	X =  325.043  mm,	Y =   -463.962  mm,	Z =   -309.100  mm,
	W =  90.000 deg,	P =   0.000 deg,	R =   90.000 deg
};
P[4144]{
   GP1:
	UF : 0, UT : 6,		CONFIG : 'N U T, 0, 0, 0',
	X =  326.503  mm,	Y =   -464.145  mm,	Z =   -309.000  mm,
	W =  90.000 deg,	P =   0.000 deg,	R =   90.000 deg
};
P[4145]{
   GP1:
	UF : 0, UT : 6,		CONFIG : 'N U T, 0, 0, 0',
	X =  326.408  mm,	Y =   -463.277  mm,	Z =   -309.100  mm,
	W =  90.000 deg,	P =   0.000 deg,	R =   90.000 deg
};
P[4146]{
   GP1:
	UF : 0, UT : 6,		CONFIG : 'N U T, 0, 0, 0',
	X =  327.820  mm,	Y =   -462.995  mm,	Z =   -314.067  mm,
	W =  90.000 deg,	P =   0.000 deg,	R =   90.000 deg
};
P[4147]{
   GP1:
	UF : 0, UT : 6,		CONFIG : 'N U T, 0, 0, 0',
	X =  329.041  mm,	Y =   -462.354  mm,	Z =   -319.718  mm,
	W =  90.000 deg,	P =   0.000 deg,	R =   90.000 deg
};
P[4148]{
   GP1:
	UF : 0, UT : 6,		CONFIG : 'N U T, 0, 0, 0',
	X =  329.280  mm,	Y =   -461.560  mm,	Z =   -309.100  mm,
	W =  90.000 deg,	P =   0.000 deg,	R =   90.000 deg
};
P[4149]{
   GP1:
	UF : 0, UT : 6,		CONFIG : 'N U T, 0, 0, 0',
	X =  330.107  mm,	Y =   -461.147  mm,	Z =   -309.100  mm,
	W =  90.000 deg,	P =   0.000 deg,	R =   90.000 deg
};
P[4150]{
   GP1:
	UF : 0, UT : 6,		CONFIG : 'N U T, 0, 0, 0',
	X =  330.865  mm,	Y =   -460.954  mm,	Z =   -309.100  mm,
	W =  90.000 deg,	P =   0.000 deg,	R =   90.000 deg
};
P[4151]{
   GP1:
	UF : 0, UT : 6,		CONFIG : 'N U T, 0, 0, 0',
	X =  332.067  mm,	Y =   -460.477  mm,	Z =   -309.050  mm,
	W =  90.000 deg,	P =   0.000 deg,	R =   90.000 deg
};
P[4152]{
   GP1:
	UF : 0, UT : 6,		CONFIG : 'N U T, 0, 0, 0',
	X =  333.038  mm,	Y =   -460.052  mm,	Z =   -320.270  mm,
	W =  90.000 deg,	P =   0.000 deg,	R =   90.000 deg
};
P[4153]{
   GP1:
	UF : 0, UT : 6,		CONFIG : 'N U T, 0, 0, 0',
	X =  333.602  mm,	Y =   -459.170  mm,	Z =   -309.000  mm,
	W =  90.000 deg,	P =   0.000 deg,	R =   90.000 deg
};
P[4154]{
   GP1:
	UF : 0, UT : 6,		CONFIG : 'N U T, 0, 0, 0',
	X =  334.380  mm,	Y =   -458.903  mm,	Z =   -318.263  mm,
	W =  90.000 deg,	P =   0.000 deg,	R =   90.000 deg
};
P[4155]{
   GP1:
	UF : 0, UT : 6,		CONFIG : 'N U T, 0, 0, 0',
	X =  335.103  mm,	Y =   -458.639  mm,	Z =   -309.100  mm,
	W =  90.000 deg,	P =   0.000 deg,	R =   90.000 deg
};
P[4156]{
   GP1:
	UF : 0, UT : 6,		CONFIG : 'N U T, 0, 0, 0',
	X =  335.858  mm,	Y =   -457.956  mm,	Z =   -309.100  mm,
	W =  90.000 deg,	P =   0.000 deg,	R =   90.000 deg
};
P[4157]{
   GP1:
	UF : 0, UT : 6,		CONFIG : 'N U T, 0, 0, 0',
	X =  337.562  mm,	Y =   -457.173  mm,	Z =   -309.100  mm,
	W =  90.000 deg,	P =   0.000 deg,	R =   90.000 deg
};
P[4158]{
   GP1:
	UF : 0, UT : 6,		CONFIG : 'N U T, 0, 0, 0',
	X =  338.604  mm,	Y =   -457.010  mm,	Z =   -313.458  mm,
	W =  90.000 deg,	P =   0.000 deg,	R =   90.000 deg
};
P[4159]{
   GP1:
	UF : 0, UT : 6,		CONFIG : 'N U T, 0, 0, 0',
	X =  339.060  mm,	Y =   -455.926  mm,	Z =   -309.100  mm,
	W =  90.000 deg,	P =   0.000 deg,	R =   90.000 deg
};
P[4160]{
   GP1:
	UF : 0, UT : 6,		CONFIG : 'N U T, 0, 0, 0',
	X =  339.781  mm,	Y =   -456.063  mm,	Z =   -325.483  mm,
	W =  90.000 deg,	P =   0.000 deg,	R =   90.000 deg
};
P[4161]{
   GP1:
	UF : 0, UT : 6,		CONFIG : 'N U T, 0, 0, 0',
	X =  340.866  mm,	Y =   -455.653  mm,	Z =   -309.100  mm,
	W =  90.000 deg,	P =   0.000 deg,	R =   90.000 deg
};
P[4162]{
   GP1:
	UF : 0, UT : 6,		CONFIG : 'N U T, 0, 0, 0',
	X =  341.602  mm,	Y =   -454.931  mm,	Z =   -309.100  mm,
	W =  90.000 deg,	P =   0.000 deg,	R =   90.000 deg
};
P[4163]{
   GP1:
	UF : 0, UT : 6,		CONFIG : 'N U T, 0, 0, 0',
	X =  342.495  mm,	Y =   -454.254  mm,	Z =   -309.100  mm,
	W =  90.000 deg,	P =   0.000 deg,	R =   90.000 deg
};
P[4164]{
   GP1:
	UF : 0, UT : 6,		CONFIG : 'N U T, 0, 0, 0',
	X =  343.799  mm,	Y =   -453.794  mm,	Z =   -316.077  mm,
	W =  90.000 deg,	P =   0.000 deg,	R =   90.000 deg
};
P[4165]{
   GP1:
	UF : 0, UT : 6,		CONFIG : 'N U T, 0, 0, 0',
	X =  344.512  mm,	Y =   -453.611  mm,	Z =   -312.115  mm,
	W =  90.000 deg,	P =   0.000 deg,	R =   90.000 deg
};
P[4166]{
   GP1:
	UF : 0, UT : 6,		CONFIG : 'N U T, 0, 0, 0',
	X =  344.893  mm,	Y =   -452.754  mm,	Z =   -309.100  mm,
	W =  90.000 deg,	P =   0.000 deg,	R =   90.000 deg
};
P[4167]{
   GP1:
	UF : 0, UT : 6,		CONFIG : 'N U T, 0, 0, 0',
	X =  345.876  mm,	Y =   -452.177  mm,	Z =   -309.100  mm,
	W =  90.000 deg,	P =   0.000 deg,	R =   90.000 deg
};
P[4168]{
   GP1:
	UF : 0, UT : 6,		CONFIG : 'N U T, 0, 0, 0',
	X =  346.784  mm,	Y =   -451.868  mm,	Z =   -317.158  mm,
	W =  90.000 deg,	P =   0.000 deg,	R =   90.000 deg
};
P[4169]{
   GP1:
	UF : 0, UT : 6,		CONFIG : 'N U T, 0, 0, 0',
	X =  347.518  mm,	Y =   -451.393  mm,	Z =   -309.100  mm,
	W =  90.000 deg,	P =   0.000 deg,	R =   90.000 deg
};
P[4170]{
   GP1:
	UF : 0, UT : 6,		CONFIG : 'N U T, 0, 0, 0',
	X =  348.500  mm,	Y =   -450.922  mm,	Z =   -309.100  mm,
	W =  90.000 deg,	P =   0.000 deg,	R =   90.000 deg
};
P[4171]{
   GP1:
	UF : 0, UT : 6,		CONFIG : 'N U T, 0, 0, 0',
	X =  349.512  mm,	Y =   -449.910  mm,	Z =   -309.100  mm,
	W =  90.000 deg,	P =   0.000 deg,	R =   90.000 deg
};
P[4172]{
   GP1:
	UF : 0, UT : 6,		CONFIG : 'N U T, 0, 0, 0',
	X =  350.498  mm,	Y =   -450.051  mm,	Z =   -317.864  mm,
	W =  90.000 deg,	P =   0.000 deg,	R =   90.000 deg
};
P[4173]{
   GP1:
	UF : 0, UT : 6,		CONFIG : 'N U T, 0, 0, 0',
	X =  351.016  mm,	Y =   -449.580  mm,	Z =   -309.100  mm,
	W =  90.000 deg,	P =   0.000 deg,	R =   90.000 deg
};
P[4174]{
   GP1:
	UF : 0, UT : 6,		CONFIG : 'N U T, 0, 0, 0',
	X =  351.932  mm,	Y =   -448.401  mm,	Z =   -309.100  mm,
	W =  90.000 deg,	P =   0.000 deg,	R =   90.000 deg
};
P[4175]{
   GP1:
	UF : 0, UT : 6,		CONFIG : 'N U T, 0, 0, 0',
	X =  352.880  mm,	Y =   -448.282  mm,	Z =   -309.100  mm,
	W =  90.000 deg,	P =   0.000 deg,	R =   90.000 deg
};
P[4176]{
   GP1:
	UF : 0, UT : 6,		CONFIG : 'N U T, 0, 0, 0',
	X =  353.986  mm,	Y =   -448.251  mm,	Z =   -325.965  mm,
	W =  90.000 deg,	P =   0.000 deg,	R =   90.000 deg
};
P[4177]{
   GP1:
	UF : 0, UT : 6,		CONFIG : 'N U T, 0, 0, 0',
	X =  354.004  mm,	Y =   -447.260  mm,	Z =   -327.146  mm,
	W =  90.000 deg,	P =   0.000 deg,	R =   90.000 deg
};
P[4178]{
   GP1:
	UF : 0, UT : 6,		CONFIG : 'N U T, 0, 0, 0',
	X =  355.173  mm,	Y =   -446.914  mm,	Z =   -309.100  mm,
	W =  90.000 deg,	P =   0.000 deg,	R =   90.000 deg
};
P[4179]{
   GP1:
	UF : 0, UT : 6,		CONFIG : 'N U T, 0, 0, 0',
	X =  356.518  mm,	Y =   -446.536  mm,	Z =   -319.705  mm,
	W =  90.000 deg,	P =   0.000 deg,	R =   90.000 deg
};
P[4180]{
   GP1:
	UF : 0, UT : 6,		CONFIG : 'N U T, 0, 0, 0',
	X =  357.300  mm,	Y =   -445.935  mm,	Z =   -309.000  mm,
	W =  90.000 deg,	P =   0.000 deg,	R =   90.000 deg
};
P[4181]{
   GP1:
	UF : 0, UT : 6,		CONFIG : 'N U T, 0, 0, 0',
	X =  358.004  mm,	Y =   -445.134  mm,	Z =   -309.100  mm,
	W =  90.000 deg,	P =   0.000 deg,	R =   90.000 deg
};
P[4182]{
   GP1:
	UF : 0, UT : 6,		CONFIG : 'N U T, 0, 0, 0',
	X =  359.292  mm,	Y =   -444.664  mm,	Z =   -309.100  mm,
	W =  90.000 deg,	P =   0.000 deg,	R =   90.000 deg
};
P[4183]{
   GP1:
	UF : 0, UT : 6,		CONFIG : 'N U T, 0, 0, 0',
	X =  360.008  mm,	Y =   -444.201  mm,	Z =   -309.000  mm,
	W =  90.000 deg,	P =   0.000 deg,	R =   90.000 deg
};
P[4184]{
   GP1:
	UF : 0, UT : 6,		CONFIG : 'N U T, 0, 0, 0',
	X =  361.188  mm,	Y =   -444.056  mm,	Z =   -325.304  mm,
	W =  90.000 deg,	P =   0.000 deg,	R =   90.000 deg
};
P[4185]{
   GP1:
	UF : 0, UT : 6,		CONFIG : 'N U T, 0, 0, 0',
	X =  361.251  mm,	Y =   -443.010  mm,	Z =   -309.000  mm,
	W =  90.000 deg,	P =   0.000 deg,	R =   90.000 deg
};
P[4186]{
   GP1:
	UF : 0, UT : 6,		CONFIG : 'N U T, 0, 0, 0',
	X =  362.524  mm,	Y =   -443.299  mm,	Z =   -325.248  mm,
	W =  90.000 deg,	P =   0.000 deg,	R =   90.000 deg
};
P[4187]{
   GP1:
	UF : 0, UT : 6,		CONFIG : 'N U T, 0, 0, 0',
	X =  363.226  mm,	Y =   -442.629  mm,	Z =   -327.645  mm,
	W =  90.000 deg,	P =   0.000 deg,	R =   90.000 deg
};
P[4188]{
   GP1:
	UF : 0, UT : 6,		CONFIG : 'N U T, 0, 0, 0',
	X =  363.688  mm,	Y =   -441.945  mm,	Z =   -309.100  mm,
	W =  90.000 deg,	P =   0.000 deg,	R =   90.000 deg
};
P[4189]{
   GP1:
	UF : 0, UT : 6,		CONFIG : 'N U T, 0, 0, 0',
	X =  370.130  mm,	Y =   -455.370  mm,	Z =   -317.842  mm,
	W =  90.000 deg,	P =   0.000 deg,	R =   90.000 deg
};
P[4190]{
   GP1:
	UF : 0, UT : 6,		CONFIG : 'N U T, 0, 0, 0',
	X =  368.313  mm,	Y =   -456.695  mm,	Z =   -320.178  mm,
	W =  90.000 deg,	P =   0.000 deg,	R =   90.000 deg
};
P[4191]{
   GP1:
	UF : 0, UT : 6,		CONFIG : 'N U T, 0, 0, 0',
	X =  367.264  mm,	Y =   -457.201  mm,	Z =   -313.957  mm,
	W =  90.000 deg,	P =   0.000 deg,	R =   90.000 deg
};
P[4192]{
   GP1:
	UF : 0, UT : 6,		CONFIG : 'N U T, 0, 0, 0',
	X =  366.190  mm,	Y =   -457.852  mm,	Z =   -309.100  mm,
	W =  90.000 deg,	P =   0.000 deg,	R =   90.000 deg
};
P[4193]{
   GP1:
	UF : 0, UT : 6,		CONFIG : 'N U T, 0, 0, 0',
	X =  365.352  mm,	Y =   -458.380  mm,	Z =   -323.127  mm,
	W =  90.000 deg,	P =   0.000 deg,	R =   90.000 deg
};
P[4194]{
   GP1:
	UF : 0, UT : 6,		CONFIG : 'N U T, 0, 0, 0',
	X =  364.251  mm,	Y =   -458.803  mm,	Z =   -313.263  mm,
	W =  90.000 deg,	P =   0.000 deg,	R =   90.000 deg
};
P[4195]{
   GP1:
	UF : 0, UT : 6,		CONFIG : 'N U T, 0, 0, 0',
	X =  362.988  mm,	Y =   -459.744  mm,	Z =   -323.904  mm,
	W =  90.000 deg,	P =   0.000 deg,	R =   90.000 deg
};
P[4196]{
   GP1:
	UF : 0, UT : 6,		CONFIG : 'N U T, 0, 0, 0',
	X =  360.054  mm,	Y =   -461.028  mm,	Z =   -309.944  mm,
	W =  90.000 deg,	P =   0.000 deg,	R =   90.000 deg
};
P[4197]{
   GP1:
	UF : 0, UT : 6,		CONFIG : 'N U T, 0, 0, 0',
	X =  359.210  mm,	Y =   -461.622  mm,	Z =   -309.000  mm,
	W =  90.000 deg,	P =   0.000 deg,	R =   90.000 deg
};
P[4198]{
   GP1:
	UF : 0, UT : 6,		CONFIG : 'N U T, 0, 0, 0',
	X =  357.631  mm,	Y =   -462.836  mm,	Z =   -323.003  mm,
	W =  90.000 deg,	P =   0.000 deg,	R =   90.000 deg
};
P[4199]{
   GP1:
	UF : 0, UT : 6,		CONFIG : 'N U T, 0, 0, 0',
	X =  356.113  mm,	Y =   -463.744  mm,	Z =   -321.634  mm,
	W =  90.000 deg,	P =   0.000 deg,	R =   90.000 deg
};
P[4200]{
   GP1:
	UF : 0, UT : 6,		CONFIG : 'N U T, 0, 0, 0',
	X =  353.522  mm,	Y =   -465.245  mm,	Z =   -309.100  mm,
	W =  90.000 deg,	P =   0.000 deg,	R =   90.000 deg
};
P[4201]{
   GP1:
	UF : 0, UT : 6,		CONFIG : 'N U T, 0, 0, 0',
	X =  352.483  mm,	Y =   -465.710  mm,	Z =   -326.795  mm,
	W =  90.000 deg,	P =   0.000 deg,	R =   90.000 deg
};
P[4202]{
   GP1:
	UF : 0, UT : 6,		CONFIG : 'N U T, 0, 0, 0',
	X =  351.674  mm,	Y =   -466.319  mm,	Z =   -318.134  mm,
	W =  90.000 deg,	P =   0.000 deg,	R =   90.000 deg
};
P[4203]{
   GP1:
	UF : 0, UT : 6,		CONFIG : 'N U T, 0, 0, 0',
	X =  350.928  mm,	Y =   -466.372  mm,	Z =   -321.296  mm,
	W =  90.000 deg,	P =   0.000 deg,	R =   90.000 deg
};
P[4204]{
   GP1:
	UF : 0, UT : 6,		CONFIG : 'N U T, 0, 0, 0',
	X =  348.318  mm,	Y =   -468.184  mm,	Z =   -326.716  mm,
	W =  90.000 deg,	P =   0.000 deg,	R =   90.000 deg
};
P[4205]{
   GP1:
	UF : 0, UT : 6,		CONFIG : 'N U T, 0, 0, 0',
	X =  347.496  mm,	Y =   -468.815  mm,	Z =   -311.962  mm,
	W =  90.000 deg,	P =   0.000 deg,	R =   90.000 deg
};
P[4206]{
   GP1:
	UF : 0, UT : 6,		CONFIG : 'N U T, 0, 0, 0',
	X =  346.336  mm,	Y =   -469.289  mm,	Z =   -312.176  mm,
	W =  90.000 deg,	P =   0.000 deg,	R =   90.000 deg
};
P[4207]{
   GP1:
	UF : 0, UT : 6,		CONFIG : 'N U T, 0, 0, 0',
	X =  345.624  mm,	Y =   -469.470  mm,	Z =   -309.000  mm,
	W =  90.000 deg,	P =   0.000 deg,	R =   90.000 deg
};
P[4208]{
   GP1:
	UF : 0, UT : 6,		CONFIG : 'N U T, 0, 0, 0',
	X =  344.976  mm,	Y =   -469.959  mm,	Z =   -312.414  mm,
	W =  90.000 deg,	P =   0.000 deg,	R =   90.000 deg
};
P[4209]{
   GP1:
	UF : 0, UT : 6,		CONFIG : 'N U T, 0, 0, 0',
	X =  344.160  mm,	Y =   -470.743  mm,	Z =   -313.140  mm,
	W =  90.000 deg,	P =   0.000 deg,	R =   90.000 deg
};
P[4210]{
   GP1:
	UF : 0, UT : 6,		CONFIG : 'N U T, 0, 0, 0',
	X =  343.250  mm,	Y =   -471.076  mm,	Z =   -309.000  mm,
	W =  90.000 deg,	P =   0.000 deg,	R =   90.000 deg
};
P[4211]{
   GP1:
	UF : 0, UT : 6,		CONFIG : 'N U T, 0, 0, 0',
	X =  342.335  mm,	Y =   -471.791  mm,	Z =   -309.100  mm,
	W =  90.000 deg,	P =   0.000 deg,	R =   90.000 deg
};
P[4212]{
   GP1:
	UF : 0, UT : 6,		CONFIG : 'N U T, 0, 0, 0',
	X =  341.451  mm,	Y =   -472.238  mm,	Z =   -309.796  mm,
	W =  90.000 deg,	P =   0.000 deg,	R =   90.000 deg
};
P[4213]{
   GP1:
	UF : 0, UT : 6,		CONFIG : 'N U T, 0, 0, 0',
	X =  340.084  mm,	Y =   -473.084  mm,	Z =   -315.122  mm,
	W =  90.000 deg,	P =   0.000 deg,	R =   90.000 deg
};
P[4214]{
   GP1:
	UF : 0, UT : 6,		CONFIG : 'N U T, 0, 0, 0',
	X =  338.651  mm,	Y =   -473.581  mm,	Z =   -314.828  mm,
	W =  90.000 deg,	P =   0.000 deg,	R =   90.000 deg
};
P[4215]{
   GP1:
	UF : 0, UT : 6,		CONFIG : 'N U T, 0, 0, 0',
	X =  337.830  mm,	Y =   -473.912  mm,	Z =   -322.397  mm,
	W =  90.000 deg,	P =   0.000 deg,	R =   90.000 deg
};
P[4216]{
   GP1:
	UF : 0, UT : 6,		CONFIG : 'N U T, 0, 0, 0',
	X =  336.722  mm,	Y =   -474.600  mm,	Z =   -315.900  mm,
	W =  90.000 deg,	P =   0.000 deg,	R =   90.000 deg
};
P[4217]{
   GP1:
	UF : 0, UT : 6,		CONFIG : 'N U T, 0, 0, 0',
	X =  335.536  mm,	Y =   -475.219  mm,	Z =   -309.100  mm,
	W =  90.000 deg,	P =   0.000 deg,	R =   90.000 deg
};
P[4218]{
   GP1:
	UF : 0, UT : 6,		CONFIG : 'N U T, 0, 0, 0',
	X =  334.878  mm,	Y =   -475.959  mm,	Z =   -326.354  mm,
	W =  90.000 deg,	P =   0.000 deg,	R =   90.000 deg
};
P[4219]{
   GP1:
	UF : 0, UT : 6,		CONFIG : 'N U T, 0, 0, 0',
	X =  333.966  mm,	Y =   -476.591  mm,	Z =   -322.102  mm,
	W =  90.000 deg,	P =   0.000 deg,	R =   90.000 deg
};
P[4220]{
   GP1:
	UF : 0, UT : 6,		CONFIG : 'N U T, 0, 0, 0',
	X =  333.254  mm,	Y =   -477.029  mm,	Z =   -309.000  mm,
	W =  90.000 deg,	P =   0.000 deg,	R =   90.000 deg
};
P[4221]{
   GP1:
	UF : 0, UT : 6,		CONFIG : 'N U T, 0, 0, 0',
	X =  330.547  mm,	Y =   -478.456  mm,	Z =   -326.060  mm,
	W =  90.000 deg,	P =   0.000 deg,	R =   90.000 deg
};
P[4222]{
   GP1:
	UF : 0, UT : 6,		CONFIG : 'N U T, 0, 0, 0',
	X =  329.060  mm,	Y =   -479.157  mm,	Z =   -313.599  mm,
	W =  90.000 deg,	P =   0.000 deg,	R =   90.000 deg
};
P[4223]{
   GP1:
	UF : 0, UT : 6,		CONFIG : 'N U T, 0, 0, 0',
	X =  327.871  mm,	Y =   -479.953  mm,	Z =   -311.541  mm,
	W =  90.000 deg,	P =   0.000 deg,	R =   90.000 deg
};
P[4224]{
   GP1:
	UF : 0, UT : 6,		CONFIG : 'N U T, 0, 0, 0',
	X =  327.272  mm,	Y =   -480.484  mm,	Z =   -327.441  mm,
	W =  90.000 deg,	P =   0.000 deg,	R =   90.000 deg
};
P[4225]{
   GP1:
	UF : 0, UT : 6,		CONFIG : 'N U T, 0, 0, 0',
	X =  325.115  mm,	Y =   -481.320  mm,	Z =   -319.370  mm,
	W =  90.000 deg,	P =   0.000 deg,	R =   90.000 deg
};
P[4226]{
   GP1:
	UF : 0, UT : 6,		CONFIG : 'N U T, 0, 0, 0',
	X =  323.945  mm,	Y =   -482.264  mm,	Z =   -323.310  mm,
	W =  90.000 deg,	P =   0.000 deg,	R =   90.000 deg
};
P[4227]{
   GP1:
	UF : 0, UT : 6,		CONFIG : 'N U T, 0, 0, 0',
	X =  323.033  mm,	Y =   -482.925  mm,	Z =   -311.088  mm,
	W =  90.000 deg,	P =   0.000 deg,	R =   90.000 deg
};
P[4228]{
   GP1:
	UF : 0, UT : 6,		CONFIG : 'N U T, 0, 0, 0',
	X =  322.353  mm,	Y =   -483.235  mm,	Z =   -319.952  mm,
	W =  90.000 deg,	P =   0.000 deg,	R =   90.000 deg
};
P[4229]{
   GP1:
	UF : 0, UT : 6,		CONFIG : 'N U T, 0, 0, 0',
	X =  321.581  mm,	Y =   -483.397  mm,	Z =   -309.100  mm,
	W =  90.000 deg,	P =   0.000 deg,	R =   90.000 deg
};
P[4230]{
   GP1:
	UF : 0, UT : 6,		CONFIG : 'N U T, 0, 0, 0',
	X =  320.384  mm,	Y =   -484.322  mm,	Z =   -323.649  mm,
	W =  90.000 deg,	P =   0.000 deg,	R =   90.000 deg
};
P[4231]{
   GP1:
	UF : 0, UT : 6,		CONFIG : 'N U T, 0, 0, 0',
	X =  318.986  mm,	Y =   -485.056  mm,	Z =   -309.000  mm,
	W =  90.000 deg,	P =   0.000 deg,	R =   90.000 deg
};
P[4232]{
   GP1:
	UF : 0, UT : 6,		CONFIG : 'N U T, 0, 0, 0',
	X =  317.976  mm,	Y =   -485.405  mm,	Z =   -321.223  mm,
	W =  90.000 deg,	P =   0.000 deg,	R =   90.000 deg
};
P[4233]{
   GP1:
	UF : 0, UT : 6,		CONFIG : 'N U T, 0, 0, 0',
	X =  317.017  mm,	Y =   -486.084  mm,	Z =   -313.401  mm,
	W =  90.000 deg,	P =   0.000 deg,	R =   90.000 deg
};
P[4234]{
   GP1:
	UF : 0, UT : 6,		CONFIG : 'N U T, 0, 0, 0',
	X =  316.577  mm,	Y =   -486.658  mm,	Z =   -313.931  mm,
	W =  90.000 deg,	P =   0.000 deg,	R =   90.000 deg
};
P[4235]{
   GP1:
	UF : 0, UT : 6,		CONFIG : 'N U T, 0, 0, 0',
	X =  315.204  mm,	Y =   -487.174  mm,	Z =   -318.974  mm,
	W =  90.000 deg,	P =   0.000 deg,	R =   90.000 deg
};
P[4236]{
   GP1:
	UF : 0, UT : 6,		CONFIG : 'N U T, 0, 0, 0',
	X =  314.075  mm,	Y =   -487.965  mm,	Z =   -323.247  mm,
	W =  90.000 deg,	P =   0.000 deg,	R =   90.000 deg
};
P[4237]{
   GP1:
	UF : 0, UT : 6,		CONFIG : 'N U T, 0, 0, 0',
	X =  312.793  mm,	Y =   -488.331  mm,	Z =   -311.315  mm,
	W =  90.000 deg,	P =   0.000 deg,	R =   90.000 deg
};
P[4238]{
   GP1:
	UF : 0, UT : 6,		CONFIG : 'N U T, 0, 0, 0',
	X =  312.228  mm,	Y =   -489.102  mm,	Z =   -311.971  mm,
	W =  90.000 deg,	P =   0.000 deg,	R =   90.000 deg
};
P[4239]{
   GP1:
	UF : 0, UT : 6,		CONFIG : 'N U T, 0, 0, 0',
	X =  311.208  mm,	Y =   -489.769  mm,	Z =   -309.100  mm,
	W =  90.000 deg,	P =   0.000 deg,	R =   90.000 deg
};
P[4240]{
   GP1:
	UF : 0, UT : 6,		CONFIG : 'N U T, 0, 0, 0',
	X =  310.069  mm,	Y =   -490.406  mm,	Z =   -322.968  mm,
	W =  90.000 deg,	P =   0.000 deg,	R =   90.000 deg
};
P[4241]{
   GP1:
	UF : 0, UT : 6,		CONFIG : 'N U T, 0, 0, 0',
	X =  307.990  mm,	Y =   -491.509  mm,	Z =   -309.000  mm,
	W =  90.000 deg,	P =   0.000 deg,	R =   90.000 deg
};
P[4242]{
   GP1:
	UF : 0, UT : 6,		CONFIG : 'N U T, 0, 0, 0',
	X =  307.080  mm,	Y =   -491.884  mm,	Z =   -317.257  mm,
	W =  90.000 deg,	P =   0.000 deg,	R =   90.000 deg
};
P[4243]{
   GP1:
	UF : 0, UT : 6,		CONFIG : 'N U T, 0, 0, 0',
	X =  306.110  mm,	Y =   -492.257  mm,	Z =   -320.855  mm,
	W =  90.000 deg,	P =   0.000 deg,	R =   90.000 deg
};
P[4244]{
   GP1:
	UF : 0, UT : 6,		CONFIG : 'N U T, 0, 0, 0',
	X =  305.486  mm,	Y =   -492.796  mm,	Z =   -324.798  mm,
	W =  90.000 deg,	P =   0.000 deg,	R =   90.000 deg
};
P[4245]{
   GP1:
	UF : 0, UT : 6,		CONFIG : 'N U T, 0, 0, 0',
	X =  304.863  mm,	Y =   -493.261  mm,	Z =   -324.523  mm,
	W =  90.000 deg,	P =   0.000 deg,	R =   90.000 deg
};
P[4246]{
   GP1:
	UF : 0, UT : 6,		CONFIG : 'N U T, 0, 0, 0',
	X =  303.709  mm,	Y =   -493.844  mm,	Z =   -324.912  mm,
	W =  90.000 deg,	P =   0.000 deg,	R =   90.000 deg
};
P[4247]{
   GP1:
	UF : 0, UT : 6,		CONFIG : 'N U T, 0, 0, 0',
	X =  302.792  mm,	Y =   -494.531  mm,	Z =   -309.100  mm,
	W =  90.000 deg,	P =   0.000 deg,	R =   90.000 deg
};
P[4248]{
   GP1:
	UF : 0, UT : 6,		CONFIG : 'N U T, 0, 0, 0',
	X =  301.496  mm,	Y =   -495.214  mm,	Z =   -324.361  mm,
	W =  90.000 deg,	P =   0.000 deg,	R =   90.000 deg
};
P[4249]{
   GP1:
	UF : 0, UT : 6,		CONFIG : 'N U T, 0, 0, 0',
	X =  300.435  mm,	Y =   -495.750  mm,	Z =   -309.000  mm,
	W =  90.000 deg,	P =   0.000 deg,	R =   90.000 deg
};
P[4250]{
   GP1:
	UF : 0, UT : 6,		CONFIG : 'N U T, 0, 0, 0',
	X =  298.649  mm,	Y =   -496.961  mm,	Z =   -312.465  mm,
	W =  90.000 deg,	P =   0.000 deg,	R =   90.000 deg
};
P[4251]{
   GP1:
	UF : 0, UT : 6,		CONFIG : 'N U T, 0, 0, 0',
	X =  297.643  mm,	Y =   -497.369  mm,	Z =   -327.276  mm,
	W =  90.000 deg,	P =   0.000 deg,	R =   90.000 deg
};
P[4252]{
   GP1:
	UF : 0, UT : 6,		CONFIG : 'N U T, 0, 0, 0',
	X =  296.699  mm,	Y =   -497.888  mm,	Z =   -325.030  mm,
	W =  90.000 deg,	P =   0.000 deg,	R =   90.000 deg
};
P[4253]{
   GP1:
	UF : 0, UT : 6,		CONFIG : 'N U T, 0, 0, 0',
	X =  296.076  mm,	Y =   -498.425  mm,	Z =   -317.421  mm,
	W =  90.000 deg,	P =   0.000 deg,	R =   90.000 deg
};
P[4254]{
   GP1:
	UF : 0, UT : 6,		CONFIG : 'N U T, 0, 0, 0',
	X =  295.262  mm,	Y =   -498.510  mm,	Z =   -327.980  mm,
	W =  90.000 deg,	P =   0.000 deg,	R =   90.000 deg
};
P[4255]{
   GP1:
	UF : 0, UT : 6,		CONFIG : 'N U T, 0, 0, 0',
	X =  294.194  mm,	Y =   -499.584  mm,	Z =   -309.568  mm,
	W =  90.000 deg,	P =   0.000 deg,	R =   90.000 deg
};
P[4256]{
   GP1:
	UF : 0, UT : 6,		CONFIG : 'N U T, 0, 0, 0',
	X =  293.467  mm,	Y =   -499.512  mm,	Z =   -323.031  mm,
	W =  90.000 deg,	P =   0.000 deg,	R =   90.000 deg
};
P[4257]{
   GP1:
	UF : 0, UT : 6,		CONFIG : 'N U T, 0, 0, 0',
	X =  291.843  mm,	Y =   -500.658  mm,	Z =   -316.063  mm,
	W =  90.000 deg,	P =   0.000 deg,	R =   90.000 deg
};
P[4258]{
   GP1:
	UF : 0, UT : 6,		CONFIG : 'N U T, 0, 0, 0',
	X =  291.061  mm,	Y =   -501.097  mm,	Z =   -310.941  mm,
	W =  90.000 deg,	P =   0.000 deg,	R =   90.000 deg
};
P[4259]{
   GP1:
	UF : 0, UT : 6,		CONFIG : 'N U T, 0, 0, 0',
	X =  289.807  mm,	Y =   -502.013  mm,	Z =   -317.383  mm,
	W =  90.000 deg,	P =   0.000 deg,	R =   90.000 deg
};
P[4260]{
   GP1:
	UF : 0, UT : 6,		CONFIG : 'N U T, 0, 0, 0',
	X =  289.052  mm,	Y =   -502.193  mm,	Z =   -313.060  mm,
	W =  90.000 deg,	P =   0.000 deg,	R =   90.000 deg
};
P[4261]{
   GP1:
	UF : 0, UT : 6,		CONFIG : 'N U T, 0, 0, 0',
	X =  288.159  mm,	Y =   -503.035  mm,	Z =   -309.000  mm,
	W =  90.000 deg,	P =   0.000 deg,	R =   90.000 deg
};
P[4262]{
   GP1:
	UF : 0, UT : 6,		CONFIG : 'N U T, 0, 0, 0',
	X =  286.879  mm,	Y =   -503.579  mm,	Z =   -327.370  mm,
	W =  90.000 deg,	P =   0.000 deg,	R =   90.000 deg
};
P[4263]{
   GP1:
	UF : 0, UT : 6,		CONFIG : 'N U T, 0, 0, 0',
	X =  285.972  mm,	Y =   -504.314  mm,	Z =   -309.100  mm,
	W =  90.000 deg,	P =   0.000 deg,	R =   90.000 deg
};
P[4264]{
   GP1:
	UF : 0, UT : 6,		CONFIG : 'N U T, 0, 0, 0',
	X =  284.922  mm,	Y =   -504.799  mm,	Z =   -309.000  mm,
	W =  90.000 deg,	P =   0.000 deg,	R =   90.000 deg
};
P[4265]{
   GP1:
	UF : 0, UT : 6,		CONFIG : 'N U T, 0, 0, 0',
	X =  283.518  mm,	Y =   -505.597  mm,	Z =   -324.774  mm,
	W =  90.000 deg,	P =   0.000 deg,	R =   90.000 deg
};
P[4266]{
   GP1:
	UF : 0, UT : 6,		CONFIG : 'N U T, 0, 0, 0',
	X =  281.621  mm,	Y =   -506.363  mm,	Z =   -322.876  mm,
	W =  90.000 deg,	P =   0.000 deg,	R =   90.000 deg
};
P[4267]{
   GP1:
	UF : 0, UT : 6,		CONFIG : 'N U T, 0, 0, 0',
	X =  280.710  mm,	Y =   -507.128  mm,	Z =   -309.000  mm,
	W =  90.000 deg,	P =   0.000 deg,	R =   90.000 deg
};
P[4268]{
   GP1:
	UF : 0, UT : 6,		CONFIG : 'N U T, 0, 0, 0',
	X =  279.612  mm,	Y =   -507.607  mm,	Z =   -319.853  mm,
	W =  90.000 deg,	P =   0.000 deg,	R =   90.000 deg
};
P[4269]{
   GP1:
	UF : 0, UT : 6,		CONFIG : 'N U T, 0, 0, 0',
	X =  278.497  mm,	Y =   -508.589  mm,	Z =   -309.000  mm,
	W =  90.000 deg,	P =   0.000 deg,	R =   90.000 deg
};
P[4270]{
   GP1:
	UF : 0, UT : 6,		CONFIG : 'N U T, 0, 0, 0',
	X =  277.085  mm,	Y =   -509.319  mm,	Z =   -326.506  mm,
	W =  90.000 deg,	P =   0.000 deg,	R =   90.000 deg
};
P[4271]{
   GP1:
	UF : 0, UT : 6,		CONFIG : 'N U T, 0, 0, 0',
	X =  275.580  mm,	Y =   -509.805  mm,	Z =   -309.992  mm,
	W =  90.000 deg,	P =   0.000 deg,	R =   90.000 deg
};
P[4272]{
   GP1:
	UF : 0, UT : 6,		CONFIG : 'N U T, 0, 0, 0',
	X =  274.490  mm,	Y =   -510.823  mm,	Z =   -309.000  mm,
	W =  90.000 deg,	P =   0.000 deg,	R =   90.000 deg
};
P[4273]{
   GP1:
	UF : 0, UT : 6,		CONFIG : 'N U T, 0, 0, 0',
	X =  273.395  mm,	Y =   -511.462  mm,	Z =   -325.321  mm,
	W =  90.000 deg,	P =   0.000 deg,	R =   90.000 deg
};
P[4274]{
   GP1:
	UF : 0, UT : 6,		CONFIG : 'N U T, 0, 0, 0',
	X =  272.390  mm,	Y =   -511.953  mm,	Z =   -327.295  mm,
	W =  90.000 deg,	P =   0.000 deg,	R =   90.000 deg
};
P[4275]{
   GP1:
	UF : 0, UT : 6,		CONFIG : 'N U T, 0, 0, 0',
	X =  271.591  mm,	Y =   -512.486  mm,	Z =   -309.100  mm,
	W =  90.000 deg,	P =   0.000 deg,	R =   90.000 deg
};
P[4276]{
   GP1:
	UF : 0, UT : 6,		CONFIG : 'N U T, 0, 0, 0',
	X =  269.800  mm,	Y =   -513.366  mm,	Z =   -309.730  mm,
	W =  90.000 deg,	P =   0.000 deg,	R =   90.000 deg
};
P[4277]{
   GP1:
	UF : 0, UT : 6,		CONFIG : 'N U T, 0, 0, 0',
	X =  268.979  mm,	Y =   -514.147  mm,	Z =   -325.756  mm,
	W =  90.000 deg,	P =   0.000 deg,	R =   90.000 deg
};
P[4278]{
   GP1:
	UF : 0, UT : 6,		CONFIG : 'N U T, 0, 0, 0',
	X =  267.638  mm,	Y =   -514.775  mm,	Z =   -309.100  mm,
	W =  90.000 deg,	P =   0.000 deg,	R =   90.000 deg
};
P[4279]{
   GP1:
	UF : 0, UT : 6,		CONFIG : 'N U T, 0, 0, 0',
	X =  264.406  mm,	Y =   -516.430  mm,	Z =   -317.911  mm,
	W =  90.000 deg,	P =   0.000 deg,	R =   90.000 deg
};
P[4280]{
   GP1:
	UF : 0, UT : 6,		CONFIG : 'N U T, 0, 0, 0',
	X =  263.386  mm,	Y =   -516.961  mm,	Z =   -320.572  mm,
	W =  90.000 deg,	P =   0.000 deg,	R =   90.000 deg
};
P[4281]{
   GP1:
	UF : 0, UT : 6,		CONFIG : 'N U T, 0, 0, 0',
	X =  261.544  mm,	Y =   -518.041  mm,	Z =   -309.000  mm,
	W =  90.000 deg,	P =   0.000 deg,	R =   90.000 deg
};
P[4282]{
   GP1:
	UF : 0, UT : 6,		CONFIG : 'N U T, 0, 0, 0',
	X =  260.714  mm,	Y =   -518.799  mm,	Z =   -309.100  mm,
	W =  90.000 deg,	P =   0.000 deg,	R =   90.000 deg
};
P[4283]{
   GP1:
	UF : 0, UT : 6,		CONFIG : 'N U T, 0, 0, 0',
	X =  259.713  mm,	Y =   -519.460  mm,	Z =   -309.000  mm,
	W =  90.000 deg,	P =   0.000 deg,	R =   90.000 deg
};
P[4284]{
   GP1:
	UF : 0, UT : 6,		CONFIG : 'N U T, 0, 0, 0',
	X =  258.056  mm,	Y =   -520.238  mm,	Z =   -318.989  mm,
	W =  90.000 deg,	P =   0.000 deg,	R =   90.000 deg
};
P[4285]{
   GP1:
	UF : 0, UT : 6,		CONFIG : 'N U T, 0, 0, 0',
	X =  256.820  mm,	Y =   -520.887  mm,	Z =   -309.100  mm,
	W =  90.000 deg,	P =   0.000 deg,	R =   90.000 deg
};
P[4286]{
   GP1:
	UF : 0, UT : 6,		CONFIG : 'N U T, 0, 0, 0',
	X =  255.528  mm,	Y =   -521.825  mm,	Z =   -322.708  mm,
	W =  90.000 deg,	P =   0.000 deg,	R =   90.000 deg
};
P[4287]{
   GP1:
	UF : 0, UT : 6,		CONFIG : 'N U T, 0, 0, 0',
	X =  254.364  mm,	Y =   -522.221  mm,	Z =   -315.447  mm,
	W =  90.000 deg,	P =   0.000 deg,	R =   90.000 deg
};
P[4288]{
   GP1:
	UF : 0, UT : 6,		CONFIG : 'N U T, 0, 0, 0',
	X =  253.809  mm,	Y =   -522.723  mm,	Z =   -324.730  mm,
	W =  90.000 deg,	P =   0.000 deg,	R =   90.000 deg
};
P[4289]{
   GP1:
	UF : 0, UT : 6,		CONFIG : 'N U T, 0, 0, 0',
	X =  251.969  mm,	Y =   -523.731  mm,	Z =   -309.100  mm,
	W =  90.000 deg,	P =   0.000 deg,	R =   90.000 deg
};
P[4290]{
   GP1:
	UF : 0, UT : 6,		CONFIG : 'N U T, 0, 0, 0',
	X =  250.489  mm,	Y =   -524.569  mm,	Z =   -325.046  mm,
	W =  90.000 deg,	P =   0.000 deg,	R =   90.000 deg
};
P[4291]{
   GP1:
	UF : 0, UT : 6,		CONFIG : 'N U T, 0, 0, 0',
	X =  249.309  mm,	Y =   -525.283  mm,	Z =   -309.100  mm,
	W =  90.000 deg,	P =   0.000 deg,	R =   90.000 deg
};
P[4292]{
   GP1:
	UF : 0, UT : 6,		CONFIG : 'N U T, 0, 0, 0',
	X =  248.209  mm,	Y =   -525.765  mm,	Z =   -316.697  mm,
	W =  90.000 deg,	P =   0.000 deg,	R =   90.000 deg
};
P[4293]{
   GP1:
	UF : 0, UT : 6,		CONFIG : 'N U T, 0, 0, 0',
	X =  247.777  mm,	Y =   -526.363  mm,	Z =   -317.984  mm,
	W =  90.000 deg,	P =   0.000 deg,	R =   90.000 deg
};
P[4294]{
   GP1:
	UF : 0, UT : 6,		CONFIG : 'N U T, 0, 0, 0',
	X =  246.576  mm,	Y =   -526.989  mm,	Z =   -320.791  mm,
	W =  90.000 deg,	P =   0.000 deg,	R =   90.000 deg
};
P[4295]{
   GP1:
	UF : 0, UT : 6,		CONFIG : 'N U T, 0, 0, 0',
	X =  245.895  mm,	Y =   -527.396  mm,	Z =   -318.034  mm,
	W =  90.000 deg,	P =   0.000 deg,	R =   90.000 deg
};
P[4296]{
   GP1:
	UF : 0, UT : 6,		CONFIG : 'N U T, 0, 0, 0',
	X =  244.727  mm,	Y =   -527.889  mm,	Z =   -325.370  mm,
	W =  90.000 deg,	P =   0.000 deg,	R =   90.000 deg
};
P[4297]{
   GP1:
	UF : 0, UT : 6,		CONFIG : 'N U T, 0, 0, 0',
	X =  244.164  mm,	Y =   -528.398  mm,	Z =   -320.420  mm,
	W =  90.000 deg,	P =   0.000 deg,	R =   90.000 deg
};
P[4298]{
   GP1:
	UF : 0, UT : 6,		CONFIG : 'N U T, 0, 0, 0',
	X =  243.223  mm,	Y =   -528.798  mm,	Z =   -309.000  mm,
	W =  90.000 deg,	P =   0.000 deg,	R =   90.000 deg
};
P[4299]{
   GP1:
	UF : 0, UT : 6,		CONFIG : 'N U T, 0, 0, 0',
	X =  241.633  mm,	Y =   -529.659  mm,	Z =   -325.176  mm,
	W =  90.000 deg,	P =   0.000 deg,	R =   90.000 deg
};
P[4300]{
   GP1:
	UF : 0, UT : 6,		CONFIG : 'N U T, 0, 0, 0',
	X =  240.399  mm,	Y =   -530.265  mm,	Z =   -311.008  mm,
	W =  90.000 deg,	P =   0.000 deg,	R =   90.000 deg
};
P[4301]{
   GP1:
	UF : 0, UT : 6,		CONFIG : 'N U T, 0, 0, 0',
	X =  239.674  mm,	Y =   -530.580  mm,	Z =   -309.000  mm,
	W =  90.000 deg,	P =   0.000 deg,	R =   90.000 deg
};
P[4302]{
   GP1:
	UF : 0, UT : 6,		CONFIG : 'N U T, 0, 0, 0',
	X =  238.263  mm,	Y =   -531.777  mm,	Z =   -320.399  mm,
	W =  90.000 deg,	P =   0.000 deg,	R =   90.000 deg
};
P[4303]{
   GP1:
	UF : 0, UT : 6,		CONFIG : 'N U T, 0, 0, 0',
	X =  236.367  mm,	Y =   -532.895  mm,	Z =   -316.696  mm,
	W =  90.000 deg,	P =   0.000 deg,	R =   90.000 deg
};
P[4304]{
   GP1:
	UF : 0, UT : 6,		CONFIG : 'N U T, 0, 0, 0',
	X =  235.311  mm,	Y =   -533.055  mm,	Z =   -309.100  mm,
	W =  90.000 deg,	P =   0.000 deg,	R =   90.000 deg
};
P[4305]{
   GP1:
	UF : 0, UT : 6,		CONFIG : 'N U T, 0, 0, 0',
	X =  234.095  mm,	Y =   -533.779  mm,	Z =   -323.976  mm,
	W =  90.000 deg,	P =   0.000 deg,	R =   90.000 deg
};
P[4306]{
   GP1:
	UF : 0, UT : 6,		CONFIG : 'N U T, 0, 0, 0',
	X =  232.905  mm,	Y =   -534.564  mm,	Z =   -319.876  mm,
	W =  90.000 deg,	P =   0.000 deg,	R =   90.000 deg
};
P[4307]{
   GP1:
	UF : 0, UT : 6,		CONFIG : 'N U T, 0, 0, 0',
	X =  232.149  mm,	Y =   -535.076  mm,	Z =   -311.832  mm,
	W =  90.000 deg,	P =   0.000 deg,	R =   90.000 deg
};
P[4308]{
   GP1:
	UF : 0, UT : 6,		CONFIG : 'N U T, 0, 0, 0',
	X =  231.583  mm,	Y =   -535.674  mm,	Z =   -317.139  mm,
	W =  90.000 deg,	P =   0.000 deg,	R =   90.000 deg
};
P[4309]{
   GP1:
	UF : 0, UT : 6,		CONFIG : 'N U T, 0, 0, 0',
	X =  230.863  mm,	Y =   -536.125  mm,	Z =   -319.168  mm,
	W =  90.000 deg,	P =   0.000 deg,	R =   90.000 deg
};
P[4310]{
   GP1:
	UF : 0, UT : 6,		CONFIG : 'N U T, 0, 0, 0',
	X =  229.871  mm,	Y =   -536.660  mm,	Z =   -319.778  mm,
	W =  90.000 deg,	P =   0.000 deg,	R =   90.000 deg
};
P[4311]{
   GP1:
	UF : 0, UT : 6,		CONFIG : 'N U T, 0, 0, 0',
	X =  228.668  mm,	Y =   -536.901  mm,	Z =   -310.087  mm,
	W =  90.000 deg,	P =   0.000 deg,	R =   90.000 deg
};
P[4312]{
   GP1:
	UF : 0, UT : 6,		CONFIG : 'N U T, 0, 0, 0',
	X =  227.800  mm,	Y =   -537.841  mm,	Z =   -315.218  mm,
	W =  90.000 deg,	P =   0.000 deg,	R =   90.000 deg
};
P[4313]{
   GP1:
	UF : 0, UT : 6,		CONFIG : 'N U T, 0, 0, 0',
	X =  226.936  mm,	Y =   -538.270  mm,	Z =   -326.982  mm,
	W =  90.000 deg,	P =   0.000 deg,	R =   90.000 deg
};
P[4314]{
   GP1:
	UF : 0, UT : 6,		CONFIG : 'N U T, 0, 0, 0',
	X =  226.294  mm,	Y =   -538.787  mm,	Z =   -312.564  mm,
	W =  90.000 deg,	P =   0.000 deg,	R =   90.000 deg
};
P[4315]{
   GP1:
	UF : 0, UT : 6,		CONFIG : 'N U T, 0, 0, 0',
	X =  225.191  mm,	Y =   -539.306  mm,	Z =   -324.794  mm,
	W =  90.000 deg,	P =   0.000 deg,	R =   90.000 deg
};
P[4316]{
   GP1:
	UF : 0, UT : 6,		CONFIG : 'N U T, 0, 0, 0',
	X =  223.701  mm,	Y =   -540.194  mm,	Z =   -319.606  mm,
	W =  90.000 deg,	P =   0.000 deg,	R =   90.000 deg
};
P[4317]{
   GP1:
	UF : 0, UT : 6,		CONFIG : 'N U T, 0, 0, 0',
	X =  222.513  mm,	Y =   -540.465  mm,	Z =   -309.000  mm,
	W =  90.000 deg,	P =   0.000 deg,	R =   90.000 deg
};
P[4318]{
   GP1:
	UF : 0, UT : 6,		CONFIG : 'N U T, 0, 0, 0',
	X =  221.288  mm,	Y =   -541.483  mm,	Z =   -320.102  mm,
	W =  90.000 deg,	P =   0.000 deg,	R =   90.000 deg
};
P[4319]{
   GP1:
	UF : 0, UT : 6,		CONFIG : 'N U T, 0, 0, 0',
	X =  219.844  mm,	Y =   -542.223  mm,	Z =   -315.006  mm,
	W =  90.000 deg,	P =   0.000 deg,	R =   90.000 deg
};
P[4320]{
   GP1:
	UF : 0, UT : 6,		CONFIG : 'N U T, 0, 0, 0',
	X =  218.928  mm,	Y =   -542.978  mm,	Z =   -324.174  mm,
	W =  90.000 deg,	P =   0.000 deg,	R =   90.000 deg
};
P[4321]{
   GP1:
	UF : 0, UT : 6,		CONFIG : 'N U T, 0, 0, 0',
	X =  218.333  mm,	Y =   -543.394  mm,	Z =   -309.100  mm,
	W =  90.000 deg,	P =   0.000 deg,	R =   90.000 deg
};
P[4322]{
   GP1:
	UF : 0, UT : 6,		CONFIG : 'N U T, 0, 0, 0',
	X =  217.057  mm,	Y =   -543.768  mm,	Z =   -309.000  mm,
	W =  90.000 deg,	P =   0.000 deg,	R =   90.000 deg
};
P[4323]{
   GP1:
	UF : 0, UT : 6,		CONFIG : 'N U T, 0, 0, 0',
	X =  215.633  mm,	Y =   -544.779  mm,	Z =   -324.940  mm,
	W =  90.000 deg,	P =   0.000 deg,	R =   90.000 deg
};
P[4324]{
   GP1:
	UF : 0, UT : 6,		CONFIG : 'N U T, 0, 0, 0',
	X =  214.248  mm,	Y =   -545.244  mm,	Z =   -323.542  mm,
	W =  90.000 deg,	P =   0.000 deg,	R =   90.000 deg
};
P[4325]{
   GP1:
	UF : 0, UT : 6,		CONFIG : 'N U T, 0, 0, 0',
	X =  213.716  mm,	Y =   -546.039  mm,	Z =   -309.000  mm,
	W =  90.000 deg,	P =   0.000 deg,	R =   90.000 deg
};
P[4326]{
   GP1:
	UF : 0, UT : 6,		CONFIG : 'N U T, 0, 0, 0',
	X =  212.826  mm,	Y =   -546.242  mm,	Z =   -312.163  mm,
	W =  90.000 deg,	P =   0.000 deg,	R =   90.000 deg
};
P[4327]{
   GP1:
	UF : 0, UT : 6,		CONFIG : 'N U T, 0, 0, 0',
	X =  211.367  mm,	Y =   -547.408  mm,	Z =   -310.887  mm,
	W =  90.000 deg,	P =   0.000 deg,	R =   90.000 deg
};
P[4328]{
   GP1:
	UF : 0, UT : 6,		CONFIG : 'N U T, 0, 0, 0',
	X =  210.093  mm,	Y =   -548.046  mm,	Z =   -318.833  mm,
	W =  90.000 deg,	P =   0.000 deg,	R =   90.000 deg
};
P[4329]{
   GP1:
	UF : 0, UT : 6,		CONFIG : 'N U T, 0, 0, 0',
	X =  208.059  mm,	Y =   -549.189  mm,	Z =   -309.100  mm,
	W =  90.000 deg,	P =   0.000 deg,	R =   90.000 deg
};
P[4330]{
   GP1:
	UF : 0, UT : 6,		CONFIG : 'N U T, 0, 0, 0',
	X =  207.291  mm,	Y =   -549.476  mm,	Z =   -317.762  mm,
	W =  90.000 deg,	P =   0.000 deg,	R =   90.000 deg
};
P[4331]{
   GP1:
	UF : 0, UT : 6,		CONFIG : 'N U T, 0, 0, 0',
	X =  205.419  mm,	Y =   -550.674  mm,	Z =   -315.072  mm,
	W =  90.000 deg,	P =   0.000 deg,	R =   90.000 deg
};
P[4332]{
   GP1:
	UF : 0, UT : 6,		CONFIG : 'N U T, 0, 0, 0',
	X =  203.976  mm,	Y =   -551.225  mm,	Z =   -309.000  mm,
	W =  90.000 deg,	P =   0.000 deg,	R =   90.000 deg
};
P[4333]{
   GP1:
	UF : 0, UT : 6,		CONFIG : 'N U T, 0, 0, 0',
	X =  203.000  mm,	Y =   -552.224  mm,	Z =   -325.611  mm,
	W =  90.000 deg,	P =   0.000 deg,	R =   90.000 deg
};
P[4334]{
   GP1:
	UF : 0, UT : 6,		CONFIG : 'N U T, 0, 0, 0',
	X =  201.563  mm,	Y =   -553.022  mm,	Z =   -309.000  mm,
	W =  90.000 deg,	P =   0.000 deg,	R =   90.000 deg
};
P[4335]{
   GP1:
	UF : 0, UT : 6,		CONFIG : 'N U T, 0, 0, 0',
	X =  200.438  mm,	Y =   -553.384  mm,	Z =   -314.016  mm,
	W =  90.000 deg,	P =   0.000 deg,	R =   90.000 deg
};
P[4336]{
   GP1:
	UF : 0, UT : 6,		CONFIG : 'N U T, 0, 0, 0',
	X =  199.706  mm,	Y =   -553.630  mm,	Z =   -321.770  mm,
	W =  90.000 deg,	P =   0.000 deg,	R =   90.000 deg
};
P[4337]{
   GP1:
	UF : 0, UT : 6,		CONFIG : 'N U T, 0, 0, 0',
	X =  199.050  mm,	Y =   -554.275  mm,	Z =   -309.100  mm,
	W =  90.000 deg,	P =   0.000 deg,	R =   90.000 deg
};
P[4338]{
   GP1:
	UF : 0, UT : 6,		CONFIG : 'N U T, 0, 0, 0',
	X =  210.000  mm,	Y =   -375.000  mm,	Z =   -250.000  mm,
	W =  90.000 deg,	P =   0.000 deg,	R =   90.000 deg
};
/END
